// TwinCAT 3 PLC project TankFuellAnlage
// ProgramVersion: 3.1.4022.1
// libraries:
//   Tc2_Standard, * (Beckhoff Automation GmbH)
//   Tc2_System, * (Beckhoff Automation GmbH)
//   Tc3_Module, * (Beckhoff Automation GmbH)
//   VisuSymbols,3.5.10.0,System
// project tree:
//   / GlobalTextList.TcGTLO, PlcTask.TcTTO (not stored), Visualization Manager.TcVMO (not stored)
//   GVLs/ DIO.TcGVL, VISU.TcGVL
//   POUs/ Simulation.TcPOU, TankFuellAnlage.TcPOU, MAIN.TcPOU
//   VISUs/ TankFuellAnlage.TcVIS
// real-time tasks:
//   TASK PlcTask: cycle T#10ms, priority 20, ADS port 350
// motion (NC):
//   TASK NC-Task 1 SAF: cycle T#2ms, priority 4, ADS port 501
//   TASK NC-Task 1 SVB: cycle T#10ms, priority 8, ADS port 511
//   AXIS Axis 1 (id 1)
//     OtherSettings: AllowMotionCmdToSlave=true
//     encoder EncType=4
//       EncPara: MaxCount=#x0000ffff
//         Inc: RefSoftSyncMask=#x0000ffff
//     drive DrvType=24
//       Analog: ScaleFactorActTorque=0.1
//       TimeComp: TaskDelayCycles=1
//     controller CtrType=1
//       CtrPara: PriorControlFactor=1
//         Observer: BandWidth=20
//   AXIS Axis 2 (id 2)
//     OtherSettings: AllowMotionCmdToSlave=true
//     encoder EncType=4
//       EncPara: MaxCount=#x0000ffff
//         Inc: RefSoftSyncMask=#x0000ffff
//     drive DrvType=24
//       Analog: ScaleFactorActTorque=0.1
//       TimeComp: TaskDelayCycles=1
//     controller CtrType=1
//       CtrPara: PriorControlFactor=1
//         Observer: BandWidth=20
//   AXIS Axis 3 (id 3)
//     OtherSettings: AllowMotionCmdToSlave=true
//     encoder EncType=4
//       EncPara: MaxCount=#x0000ffff
//     drive DrvType=23
//       Analog: ScaleFactorActTorque=0.1
//       TimeComp: TaskDelayCycles=1
//     controller CtrType=1
//       CtrPara: PriorControlFactor=1
//         Observer: BandWidth=20
//   AXIS Axis 4 (id 4)
//     OtherSettings: AllowMotionCmdToSlave=true
//     encoder EncType=4
//       EncPara: MaxCount=#x0000ffff
//     drive DrvType=23
//       Analog: ScaleFactorActTorque=0.1
//       TimeComp: TaskDelayCycles=1
//     controller CtrType=1
//       CtrPara: PriorControlFactor=1
//         Observer: BandWidth=20
//   AXIS Axis 5 (id 5)
//     OtherSettings: AllowMotionCmdToSlave=true
//     encoder EncType=19
//       EncPara: MaxCount=#xffffffff
//     drive DrvType=16
//       DrvPara: MaxCount=#xffffffff
//         Analog: ScaleFactorActTorque=0.1
//         TimeComp: TaskDelayCycles=1
//     controller CtrType=1
//       CtrPara: PriorControlFactor=1
//         Observer: BandWidth=20
//   AXIS Axis 6 (id 6)
//     OtherSettings: AllowMotionCmdToSlave=true
//     encoder EncType=19
//       EncPara: MaxCount=#xffffffff
//     drive DrvType=16
//       DrvPara: MaxCount=#xffffffff
//         Analog: ScaleFactorActTorque=0.1
//         TimeComp: TaskDelayCycles=1
//     controller CtrType=1
//       CtrPara: PriorControlFactor=1
//         Observer: BandWidth=20
// I/O:
//   DEVICE Device 1 (EtherCAT), AmsNetId 5.35.139.20.2.1
//     Term 1 (EK1200) [EK1200-5000 EtherCAT Power supply (2A E-Bus)]
//       Term 2 (EL1809) [EL1809 16Ch. Dig. Input 24V, 3ms]
//       Term 3 (EL1809) [EL1809 16Ch. Dig. Input 24V, 3ms]
//       Term 4 (EL2809) [EL2809 16Ch. Dig. Output 24V, 0.5A]
//       Term 5 (EL2809) [EL2809 16Ch. Dig. Output 24V, 0.5A]
//       Term 6 (EL3064) [EL3064 4Ch. Ana. Input 0-10V]
//       Term 7 (EL4034) [EL4034 4Ch. Ana. Output +/-10V, 12bit]
//       Term 8 (EL7031) [EL7031 1Ch. Stepper motor output stage (24V, 1.5A)]
//       Term 9 (EL7031) [EL7031 1Ch. Stepper motor output stage (24V, 1.5A)]
//       Term 10 (EL7332) [EL7332 2Ch. DC motor output stage (24V, 1.5A)]
//       Term 11 (EL7201-0010) [EL7201-0010 1Ch. MDP742 Servo motor output stage with OCT (50V, 4A)]
//       Term 12 (EL7201-0010) [EL7201-0010 1Ch. MDP742 Servo motor output stage with OCT (50V, 4A)]
//       Term 26 (EL6090) [EL6090 Display terminal]
//       Term 27 (EK1110) [EK1110 EtherCAT extension]
// variable links:
//   NC-Task 1 SAF/Axes/Axis 1 <-> Device 1 (EtherCAT)/Term 1 (EK1200)/Term 8 (EL7031)
//     Drive/Inputs/In/nState1 @bit 3 <-> STM Status/Status/Error
//     Drive/Inputs/In/nState1 @bit 5 <-> STM Status/Status/Moving negative
//     Drive/Inputs/In/nState1 @bit 4 <-> STM Status/Status/Moving positive
//     Drive/Inputs/In/nState1 @bit 1 <-> STM Status/Status/Ready
//     Drive/Inputs/In/nState1 <-> STM Status/Status/Ready to enable
//     Drive/Inputs/In/nState1 @bit 6 <-> STM Status/Status/Torque reduced
//     Drive/Inputs/In/nState1 @bit 2 <-> STM Status/Status/Warning
//     Drive/Inputs/In/nState2 @bit 3 <-> STM Status/Status/Digital input 1
//     Drive/Inputs/In/nState2 @bit 4 <-> STM Status/Status/Digital input 2
//     Drive/Inputs/In/nState2 @bit 5 <-> STM Status/Status/Sync error
//     Drive/Inputs/In/nState2 @bit 7 <-> STM Status/Status/TxPDO Toggle
//     Drive/Inputs/In/nState4 @bit 1 <-> WcState/InputToggle
//     Drive/Inputs/In/nState4 <-> WcState/WcState
//     Drive/Outputs/Out/nCtrl1 <-> STM Control/Control/Enable
//     Drive/Outputs/Out/nCtrl1 @bit 2 <-> STM Control/Control/Reduce torque
//     Drive/Outputs/Out/nCtrl1 @bit 1 <-> STM Control/Control/Reset
//     Drive/Outputs/Out/nDataOut2[0] <-> STM Velocity/Velocity
//     Enc/Inputs/In/nDataIn1[0] <-> ENC Status compact/Counter value
//     Enc/Inputs/In/nDataIn2[0] <-> ENC Status compact/Latch value
//     Enc/Inputs/In/nState1 @bit 4 <-> ENC Status compact/Status/Counter overflow
//     Enc/Inputs/In/nState1 @bit 3 <-> ENC Status compact/Status/Counter underflow
//     Enc/Inputs/In/nState1 @bit 1 <-> ENC Status compact/Status/Latch extern valid
//     Enc/Inputs/In/nState1 @bit 2 <-> ENC Status compact/Status/Set counter done
//     Enc/Inputs/In/nState2 @bit 4 <-> ENC Status compact/Status/Status of extern latch
//     Enc/Inputs/In/nState2 @bit 5 <-> ENC Status compact/Status/Sync error
//     Enc/Inputs/In/nState2 @bit 7 <-> ENC Status compact/Status/TxPDO Toggle
//     Enc/Inputs/In/nState4 @bit 1 <-> WcState/InputToggle
//     Enc/Inputs/In/nState4 <-> WcState/WcState
//     Enc/Outputs/Out/nCtrl1 @bit 3 <-> ENC Control compact/Control/Enable latch extern on negative edge
//     Enc/Outputs/Out/nCtrl1 @bit 1 <-> ENC Control compact/Control/Enable latch extern on positive edge
//     Enc/Outputs/Out/nCtrl1 @bit 2 <-> ENC Control compact/Control/Set counter
//     Enc/Outputs/Out/nDataOut1[0] <-> ENC Control compact/Set counter value
//   NC-Task 1 SAF/Axes/Axis 2 <-> Device 1 (EtherCAT)/Term 1 (EK1200)/Term 9 (EL7031)
//     Drive/Inputs/In/nState1 @bit 3 <-> STM Status/Status/Error
//     Drive/Inputs/In/nState1 @bit 5 <-> STM Status/Status/Moving negative
//     Drive/Inputs/In/nState1 @bit 4 <-> STM Status/Status/Moving positive
//     Drive/Inputs/In/nState1 @bit 1 <-> STM Status/Status/Ready
//     Drive/Inputs/In/nState1 <-> STM Status/Status/Ready to enable
//     Drive/Inputs/In/nState1 @bit 6 <-> STM Status/Status/Torque reduced
//     Drive/Inputs/In/nState1 @bit 2 <-> STM Status/Status/Warning
//     Drive/Inputs/In/nState2 @bit 3 <-> STM Status/Status/Digital input 1
//     Drive/Inputs/In/nState2 @bit 4 <-> STM Status/Status/Digital input 2
//     Drive/Inputs/In/nState2 @bit 5 <-> STM Status/Status/Sync error
//     Drive/Inputs/In/nState2 @bit 7 <-> STM Status/Status/TxPDO Toggle
//     Drive/Inputs/In/nState4 @bit 1 <-> WcState/InputToggle
//     Drive/Inputs/In/nState4 <-> WcState/WcState
//     Drive/Outputs/Out/nCtrl1 <-> STM Control/Control/Enable
//     Drive/Outputs/Out/nCtrl1 @bit 2 <-> STM Control/Control/Reduce torque
//     Drive/Outputs/Out/nCtrl1 @bit 1 <-> STM Control/Control/Reset
//     Drive/Outputs/Out/nDataOut2[0] <-> STM Velocity/Velocity
//     Enc/Inputs/In/nDataIn1[0] <-> ENC Status compact/Counter value
//     Enc/Inputs/In/nDataIn2[0] <-> ENC Status compact/Latch value
//     Enc/Inputs/In/nState1 @bit 4 <-> ENC Status compact/Status/Counter overflow
//     Enc/Inputs/In/nState1 @bit 3 <-> ENC Status compact/Status/Counter underflow
//     Enc/Inputs/In/nState1 @bit 1 <-> ENC Status compact/Status/Latch extern valid
//     Enc/Inputs/In/nState1 @bit 2 <-> ENC Status compact/Status/Set counter done
//     Enc/Inputs/In/nState2 @bit 4 <-> ENC Status compact/Status/Status of extern latch
//     Enc/Inputs/In/nState2 @bit 5 <-> ENC Status compact/Status/Sync error
//     Enc/Inputs/In/nState2 @bit 7 <-> ENC Status compact/Status/TxPDO Toggle
//     Enc/Inputs/In/nState4 @bit 1 <-> WcState/InputToggle
//     Enc/Inputs/In/nState4 <-> WcState/WcState
//     Enc/Outputs/Out/nCtrl1 @bit 3 <-> ENC Control compact/Control/Enable latch extern on negative edge
//     Enc/Outputs/Out/nCtrl1 @bit 1 <-> ENC Control compact/Control/Enable latch extern on positive edge
//     Enc/Outputs/Out/nCtrl1 @bit 2 <-> ENC Control compact/Control/Set counter
//     Enc/Outputs/Out/nDataOut1[0] <-> ENC Control compact/Set counter value
//   NC-Task 1 SAF/Axes/Axis 3 <-> Device 1 (EtherCAT)/Term 1 (EK1200)/Term 10 (EL7332)
//     Drive/Inputs/In/nState1 @bit 3 <-> DCM Status Channel 1/Status/Error
//     Drive/Inputs/In/nState1 @bit 5 <-> DCM Status Channel 1/Status/Moving negative
//     Drive/Inputs/In/nState1 @bit 4 <-> DCM Status Channel 1/Status/Moving positive
//     Drive/Inputs/In/nState1 @bit 1 <-> DCM Status Channel 1/Status/Ready
//     Drive/Inputs/In/nState1 <-> DCM Status Channel 1/Status/Ready to enable
//     Drive/Inputs/In/nState1 @bit 6 <-> DCM Status Channel 1/Status/Torque reduced
//     Drive/Inputs/In/nState1 @bit 2 <-> DCM Status Channel 1/Status/Warning
//     Drive/Inputs/In/nState2 @bit 3 <-> DCM Status Channel 1/Status/Digital input 1
//     Drive/Inputs/In/nState2 @bit 4 <-> DCM Status Channel 1/Status/Digital input 2
//     Drive/Inputs/In/nState2 @bit 5 <-> DCM Status Channel 1/Status/Sync error
//     Drive/Inputs/In/nState2 @bit 7 <-> DCM Status Channel 1/Status/TxPDO Toggle
//     Drive/Inputs/In/nState4 @bit 1 <-> WcState/InputToggle
//     Drive/Inputs/In/nState4 <-> WcState/WcState
//     Drive/Outputs/Out/nCtrl1 <-> DCM Control Channel 1/Control/Enable
//     Drive/Outputs/Out/nCtrl1 @bit 2 <-> DCM Control Channel 1/Control/Reduce torque
//     Drive/Outputs/Out/nCtrl1 @bit 1 <-> DCM Control Channel 1/Control/Reset
//     Drive/Outputs/Out/nDataOut2[0] <-> DCM Velocity Channel 1/Velocity
//   NC-Task 1 SAF/Axes/Axis 4 <-> Device 1 (EtherCAT)/Term 1 (EK1200)/Term 10 (EL7332)
//     Drive/Inputs/In/nState1 @bit 3 <-> DCM Status Channel 2/Status/Error
//     Drive/Inputs/In/nState1 @bit 5 <-> DCM Status Channel 2/Status/Moving negative
//     Drive/Inputs/In/nState1 @bit 4 <-> DCM Status Channel 2/Status/Moving positive
//     Drive/Inputs/In/nState1 @bit 1 <-> DCM Status Channel 2/Status/Ready
//     Drive/Inputs/In/nState1 <-> DCM Status Channel 2/Status/Ready to enable
//     Drive/Inputs/In/nState1 @bit 6 <-> DCM Status Channel 2/Status/Torque reduced
//     Drive/Inputs/In/nState1 @bit 2 <-> DCM Status Channel 2/Status/Warning
//     Drive/Inputs/In/nState2 @bit 3 <-> DCM Status Channel 2/Status/Digital input 1
//     Drive/Inputs/In/nState2 @bit 4 <-> DCM Status Channel 2/Status/Digital input 2
//     Drive/Inputs/In/nState2 @bit 5 <-> DCM Status Channel 2/Status/Sync error
//     Drive/Inputs/In/nState2 @bit 7 <-> DCM Status Channel 2/Status/TxPDO Toggle
//     Drive/Inputs/In/nState4 @bit 1 <-> WcState/InputToggle
//     Drive/Inputs/In/nState4 <-> WcState/WcState
//     Drive/Outputs/Out/nCtrl1 <-> DCM Control Channel 2/Control/Enable
//     Drive/Outputs/Out/nCtrl1 @bit 2 <-> DCM Control Channel 2/Control/Reduce torque
//     Drive/Outputs/Out/nCtrl1 @bit 1 <-> DCM Control Channel 2/Control/Reset
//     Drive/Outputs/Out/nDataOut2[0] <-> DCM Velocity Channel 2/Velocity
//   NC-Task 1 SAF/Axes/Axis 5 <-> Device 1 (EtherCAT)/Term 1 (EK1200)/Term 11 (EL7201-0010)
//     Drive/Inputs/In/nDcOutputTime <-> InfoData/DcOutputShift
//     Drive/Inputs/In/nState1 <-> DRV Statusword/Statusword
//     Drive/Inputs/In/nState2 <-> DRV Statusword/Statusword @bit 8
//     Drive/Inputs/In/nState4 @bit 1 <-> WcState/InputToggle
//     Drive/Inputs/In/nState4 <-> WcState/WcState
//     Drive/Outputs/Out/nCtrl1 <-> DRV Controlword/Controlword
//     Drive/Outputs/Out/nCtrl2 <-> DRV Controlword/Controlword @bit 8
//     Drive/Outputs/Out/nDataOut2 <-> DRV Target velocity/Target velocity
//     Enc/Inputs/In/nDataIn1 <-> FB Position/Position
//     Enc/Inputs/In/nDcInputTime <-> InfoData/DcInputShift
//     Enc/Inputs/In/nState4 @bit 1 <-> WcState/InputToggle
//     Enc/Inputs/In/nState4 <-> WcState/WcState
//   NC-Task 1 SAF/Axes/Axis 6 <-> Device 1 (EtherCAT)/Term 1 (EK1200)/Term 12 (EL7201-0010)
//     Drive/Inputs/In/nDcOutputTime <-> InfoData/DcOutputShift
//     Drive/Inputs/In/nState1 <-> DRV Statusword/Statusword
//     Drive/Inputs/In/nState2 <-> DRV Statusword/Statusword @bit 8
//     Drive/Inputs/In/nState4 @bit 1 <-> WcState/InputToggle
//     Drive/Inputs/In/nState4 <-> WcState/WcState
//     Drive/Outputs/Out/nCtrl1 <-> DRV Controlword/Controlword
//     Drive/Outputs/Out/nCtrl2 <-> DRV Controlword/Controlword @bit 8
//     Drive/Outputs/Out/nDataOut2 <-> DRV Target velocity/Target velocity
//     Enc/Inputs/In/nDataIn1 <-> FB Position/Position
//     Enc/Inputs/In/nDcInputTime <-> InfoData/DcInputShift
//     Enc/Inputs/In/nState4 @bit 1 <-> WcState/InputToggle
//     Enc/Inputs/In/nState4 <-> WcState/WcState
//   TankFuellAnlage/TankFuellAnlage Instance <-> Device 1 (EtherCAT)/Term 1 (EK1200)/Term 5 (EL2809)
//     PlcTask Outputs/DIO.P1 <-> Channel 4/Output
//     PlcTask Outputs/DIO.Q1 <-> Channel 1/Output
//     PlcTask Outputs/DIO.Q2 <-> Channel 2/Output
//     PlcTask Outputs/DIO.Q3 <-> Channel 3/Output

// ---- GVLs/DIO.TcGVL
{attribute 'qualified_only'}
VAR_GLOBAL
	// Ventil für Tank 1
	Q1 AT %Q*: BOOL; 
	// Ventil für Tank 2
	Q2 AT %Q*: BOOL; 	
	// Ventil für Tank 3
	Q3 AT %Q*: BOOL; 	
	// Meldeleuchte Störung
	P1 AT %Q*: BOOL;
END_VAR

// ---- GVLs/VISU.TcGVL
{attribute 'qualified_only'}
VAR_GLOBAL
	// Schwimmerschalter Tank 1 - Leer
	B1 : BOOL; 
	// Schwimmerschalter Tank 1 - Voll
	B2 : BOOL; 
	// Schwimmerschalter Tank 2 - Leer
	B3 : BOOL; 
	// Schwimmerschalter Tank 2 - Voll
	B4 : BOOL; 
	// Schwimmerschalter Tank 3 - Leer
	B5 : BOOL; 
	// Schwimmerschalter Tank 3 - Voll
	B6 : BOOL; 	
END_VAR

// ---- POUs/Simulation.TcPOU
FUNCTION_BLOCK Simulation
VAR_INPUT
END_VAR
VAR_OUTPUT
END_VAR
VAR
	tonTaktgeber: ton;	

	xAuslass1: BOOL;	//Es wird Wasser abgelassen
	xAuslass2: BOOL;
	xAuslass3: BOOL;

	uiFuellstandTank1: UINT;	// 0 --> voll; 300 --> leer
	uiFuellstandTank2: UINT;
	uiFuellstandTank3: UINT;	
END_VAR

//Simulation für die Visualisierung
tonTaktgeber(IN:= NOT tonTaktgeber.Q, PT:= T#30MS);

IF tonTaktgeber.Q THEN
	// damit das Simulation mit passabler Geschwindigkeit läuft	

	// Tank leeren
	IF  xAuslass1 THEN
		IF uiFuellstandTank1 < 300 THEN
			uiFuellstandTank1 := uiFuellstandTank1 + 1;
		ELSE
			uiFuellstandTank1 := 300;		
		END_IF
	END_IF

	IF  xAuslass2 THEN
		IF uiFuellstandTank2 < 300 THEN
			uiFuellstandTank2 := uiFuellstandTank2 + 1;
		ELSE
			uiFuellstandTank2 := 300;		
		END_IF
	END_IF

	IF  xAuslass3 THEN
		IF uiFuellstandTank3 < 300 THEN
			uiFuellstandTank3 := uiFuellstandTank3 + 1;
		ELSE
			uiFuellstandTank3 := 300;		
		END_IF
	END_IF
	
	// Tank füllen
	IF DIO.Q1 THEN
		IF uiFuellstandTank1 > 2 THEN
			uiFuellstandTank1 := uiFuellstandTank1 - 2;
		ELSE
			uiFuellstandTank1 := 0;	
		END_IF
	END_IF
	
	IF DIO.Q2 THEN
		IF uiFuellstandTank2 > 2 THEN
			uiFuellstandTank2 := uiFuellstandTank2 - 2;
		ELSE
			uiFuellstandTank2 := 0;	
		END_IF
	END_IF
	
	IF DIO.Q3 THEN
		IF uiFuellstandTank3 > 2 THEN
			uiFuellstandTank3 := uiFuellstandTank3 - 2;
		ELSE
			uiFuellstandTank3 := 0;	
		END_IF
	END_IF
	
END_IF


// Füllstand unten
IF uiFuellstandTank1 > 290 THEN
	VISU.B1 := TRUE;
ELSE
	VISU.B1 := FALSE;
END_IF

IF uiFuellstandTank2 > 290 THEN
	VISU.B3 := TRUE;
ELSE
	VISU.B3 := FALSE;
END_IF

IF uiFuellstandTank3 > 290 THEN
	VISU.B5 := TRUE;
ELSE
	VISU.B5 := FALSE;
END_IF


// Füllstand oben
IF uiFuellstandTank1 < 10 THEN
	VISU.B2 := TRUE;
ELSE
	VISU.B2 := FALSE;
END_IF

IF uiFuellstandTank2 < 10 THEN
	VISU.B4 := TRUE;
ELSE
	VISU.B4 := FALSE;
END_IF

IF uiFuellstandTank3 < 10 THEN
	VISU.B6 := TRUE;
ELSE
	VISU.B6 := FALSE;
END_IF

END_FUNCTION_BLOCK

// ---- POUs/TankFuellAnlage.TcPOU
FUNCTION_BLOCK TankFuellAnlage
VAR_INPUT
END_VAR
VAR_OUTPUT
END_VAR
VAR
END_VAR

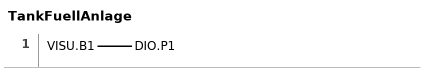
// NETWORK 1
DIO.P1 := VISU.B1;

END_FUNCTION_BLOCK

// ---- POUs/MAIN.TcPOU
PROGRAM MAIN
VAR
	TankFuellAnlage: TankFuellAnlage;
	Simulation: Simulation;
END_VAR

TankFuellAnlage();
Simulation();

END_PROGRAM

// ---- GlobalTextList.TcGTLO
TEXTLIST GlobalTextList
  410 = '-B1'
  235 = '-B2'
  26 = '-B3'
  878 = '-B4'
  946 = '-B5'
  390 = '-B6'
  88 = '-Q1'
  726 = '-Q2'
  710 = '-Q3'
  546 = '-Y1'
  973 = 'Auslass'
  141 = 'B2'
  136 = 'Lüfter 1'
  438 = 'Lüfter 2'
  522 = 'Lüfter 3'
  25 = 'Lüfter 4'
  958 = 'Tank 1'
  630 = 'Tank 2'
  349 = 'Tank 3'
END_TEXTLIST

// ---- VISUs/TankFuellAnlage.TcVIS
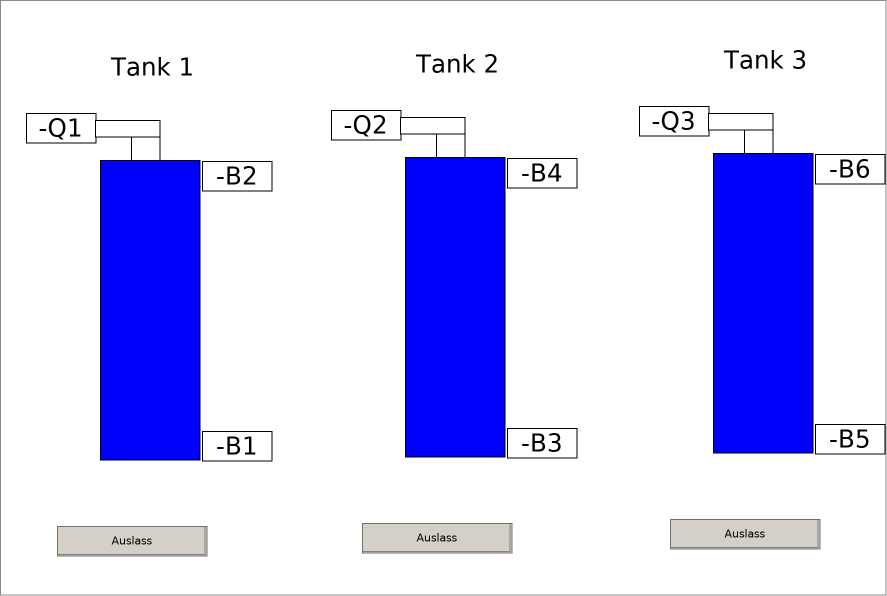
VISUALIZATION TankFuellAnlage  // 887x596
    Rectangle (128,461 29x133), colour toggle: MAIN.Simulation.xAuslass1
    Rectangle (131,120 29x305), colour toggle: DIO.Q1
    Rectangle (100,160 100x300)
    Rectangle (100,160 100x300)
        p2773130477: MAIN.Simulation.uiFuellstandTank1
    Label (105,52 95x30), "Tank 1"
    Button (57,526 150x30), "Auslass"
        tap MAIN.Simulation.xAuslass1
    Rectangle (202,161 70x30), "-B2", colour toggle: VISU.B2
    Rectangle (202,431 70x30), "-B1", colour toggle: VISU.B1
    Rectangle (26,113 70x30), "-Q1", colour toggle: DIO.Q1
    Rectangle (95,120 65x17), colour toggle: DIO.Q1
    Rectangle (436,117 29x305), colour toggle: DIO.Q2
    Rectangle (405,157 100x300)
    Rectangle (405,157 100x300)
        p2773130477: MAIN.Simulation.uiFuellstandTank2
    Label (410,49 95x30), "Tank 2"
    Button (362,523 150x30), "Auslass"
        tap MAIN.Simulation.xAuslass2
    Rectangle (507,158 70x30), "-B4", colour toggle: VISU.B4
    Rectangle (507,428 70x30), "-B3", colour toggle: VISU.B3
    Rectangle (331,110 70x30), "-Q2", colour toggle: DIO.Q2
    Rectangle (400,117 65x17), colour toggle: DIO.Q2
    Rectangle (391,183 29x301), colour toggle: DIO.Q1
    Rectangle (744,113 29x305), colour toggle: DIO.Q3
    Rectangle (713,153 100x300)
    Rectangle (713,153 100x300)
        p2773130477: MAIN.Simulation.uiFuellstandTank3
    Label (718,45 95x30), "Tank 3"
    Button (670,519 150x30), "Auslass"
        tap MAIN.Simulation.xAuslass3
    Rectangle (815,154 70x30), "-B6", colour toggle: VISU.B6
    Rectangle (815,424 70x30), "-B5", colour toggle: VISU.B5
    Rectangle (639,106 70x30), "-Q3", colour toggle: DIO.Q3
    Rectangle (708,113 65x17), colour toggle: DIO.Q3
    Rectangle (699,179 29x301), colour toggle: DIO.Q1
    Rectangle (132,150 29x305), colour toggle: DIO.Q1
    Rectangle (436,151 29x305), colour toggle: DIO.Q2
    Rectangle (747,151 29x305), colour toggle: DIO.Q3
    Rectangle (437,458 29x133), colour toggle: MAIN.Simulation.xAuslass2
    Rectangle (749,455 29x133), colour toggle: MAIN.Simulation.xAuslass3
END_VISUALIZATION
